Staubli VAL3: home.pjx

--- home.pjx ---
Parameters version=s7.2.1 stackSize=5000 millimeterUnit=true
Program file=changeSession.pgx
Program file=copy_folder.pgx
Program file=isSessionFound.pgx
Program file=loadPage.pgx
Program file=main.pgx
Program file=onEnterEvent.pgx
Program file=onExit.pgx
Program file=onF1Event.pgx
Program file=onF2Event.pgx
Program file=onF3Event.pgx
Program file=onF4Event.pgx
Program file=onF5Event.pgx
Program file=onF6Event.pgx
Program file=onF7Event.pgx
Program file=onF8Event.pgx
Program file=onStart.pgx
Program file=passwd.pgx
Program file=refresh.pgx
Program file=refreshDynamic.pgx
Program file=refreshStatic.pgx
Data file=home.dtx
Library alias=use path=Disk://kernel/userPage/userPage.pjx
Library alias=saveData path=Disk://saveData/saveData.pjx
Library alias=page path=Disk://kernel/template/page/page.pjx
Library alias=language path=Disk://kernel/language/language.pjx
Library alias=processList path=Disk://kernel/processList/processList.pjx
Library alias=cycleStatus path=Disk://cycleStatus/cycleStatus.pjx

--- home.dtx ---
num nKey = 271
public num nPage = 10
num nRefresh = 33.117
num nTime = 1
num nValue[4]
  [0] = 1
  [1] = 2
  [2] = 3
  [3] = 4
public string sItems
string sMenu
string sMessage
string sVersion = "valClean 7.3.1.8"
string sMenu8[8]
string sSession
string sPathSession
string sDeeperSession
bool bButton[8]
  [0] = true
  [1] = true
  [2] = true
  [4] = true
  [5] = true
  [6] = true
  [7] = true

--- main.pgx ---
public program main()
  local bool l_bExit
begin
  // INIT
  call onStart()
  // LOOP UNTIL Exit
  l_bExit=false
  do
    // call the refresh
    call refresh()
    // take the key
    nKey=getKey()
    switch nKey
      case 271
        // select program
        call onF1Event()
      break
      case 272
        // input output
        call onF2Event()
      break
      case 273
        // preset
        call onF3Event()
      break
      case 274
        call onF4Event()
      break
      case 275
        // production page
        call onF5Event()
      break
      case 276
        // maintenance
        call onF6Event()
      break
      case 277
        // advance
        call onF7Event()
      break
      case 278
        // exit
        call onF8Event(l_bExit)
      break
      case 270
        call onEnterEvent()
      break
    endSwitch
    //release the resource
    delay(0)
    // check for the resetMOtion
    if !cycleStatus:bCycle and !cycleStatus:bSimulation and !isEmpty()
      //resetMotion()
    endIf
  until l_bExit
  // on Exit
  call onExit()
end

--- changeSession.pgx ---
program changeSession()
  local num l_nIndex
  local num l_nSize
  local bool l_bDone
  local num i
  local num l_nResult
  local string l_sMessage
  local string l_sPaste
  local string l_sEvent
  local string l_sEmpty
  local string l_sSession
  local string l_sButton[2]
  local bool l_bOk
begin
  // init
  //
  // CREATE THE LIST
  //
  // define your list size for default
  // init
  use:nView=0
  do
    //
    cls()
    call use:setSizeList(19,0,19,11)
    call use:setView(false)
    //
    call use:listcreate("Session")
    // show the message
    call language:page(l_sMessage,1030)
    call use:stringToArray(l_sMessage,sMenu)
    sMenu=""
    if saveData:mode==1
      sMenu[6]=""
    endIf
    if saveData:mode>=1
      call use:setMenu(sMenu,true,3)
    endIf
    // clean the string
    l_sEmpty=""
    call use:stringCopy(l_sEmpty,sSession)
    // get the list of session
    call saveData:getListSession(sSession)
    // build the list
    call use:listadd(sSession)
    // update
    call use:listupdate(0)
    // read the list
    l_bDone=false
    do
      // get the item
      nKey=get()
      call use:listevent(nKey,l_nIndex,l_sEvent)
    until nKey==270 or nKey==255 or ((nKey<=278 and nKey>=275)and sMenu[nKey-271]!="")
    //
    switch nKey
      case 275
        // rename
        l_sPaste=l_sEvent
        call isSessionFound(l_sPaste,l_nResult)
        if l_sPaste!="" and l_sPaste!=l_sEvent
          $rename("session/"+l_sEvent,"session/"+l_sPaste)
        endIf
      break
      case 276
        // duplicate
        l_sPaste=l_sEvent
        call isSessionFound(l_sPaste,l_nResult)
        if l_nResult!=-1
          // duplicate all the file
          call copy_folder(l_sEvent,l_sPaste)
          l_bDone=true
        endIf
      break
      case 277
        // delete
        call saveData:getSession(l_sSession)
        if l_sEvent!=l_sSession and l_sEvent!="default"
          // delete
          call language:getYesNo(l_sButton)
          call language:message(l_sMessage,80)
          l_sMessage=l_sMessage+l_sEvent
          call use:yes_no(l_sMessage,l_sButton,l_bOk)
          if l_bOk
            $delete("Disk://session/"+l_sEvent)
          endIf
        else
          call language:message(l_sMessage,23)
          l_sMessage=l_sMessage+l_sEvent
          popUpMsg(l_sMessage)
        endIf
      break
      case 278
        // create a new one
        // look inside
        call isSessionFound(l_sPaste,l_nResult)
        if l_nResult!=-1
          // create a new one
          call copy_folder("",l_sPaste)
        endIf
      break
    endSwitch
  until l_bDone or nKey==255 or nKey==270
  //
  if nKey!=255 and cycleStatus:bCycle==false and cycleStatus:bSimulation==false
    // check if l_sPaste has been used
    if l_sPaste!=""
      l_sEvent=l_sPaste
    endIf
    // change session
    call language:message(l_sMessage,19)
    l_sMessage=l_sMessage+" SESSION DATA..."
    call use:timerDialog(l_sMessage,0)
      // load the new session
    call saveData:changeSession(l_sEvent)
    // reload the processList using the default saveCycle
    call processList:loadProcessList(i)
    // reset the homing trajectory
    cycleStatus:bHomeLoaded=false
    // save the session
    saveData:libSave()
  endIf
  //
  call use:nullKey(nKey)
end

--- copy_folder.pgx ---
program copy_folder(string x_sPathCopy, string x_sPathPaste)
  local string l_sPathCopy
  local string l_sPathPaste
  local bool l_bCheck
  local num i
  local num j
  local string l_sEmpty
begin
  //
  // copy or not the x_sPathCopy to x_sPath
  //
  call use:timerDialog("Copying file: ##",0)
  call use:stringCopy(l_sEmpty,sPathSession)
  // all the folder are created
  if x_sPathCopy==""
    // copy from the template session
    l_sPathCopy="Disk://kernel/template/session/"
  else
    // copy form the x_sPathCopy session name
    l_sPathCopy="Disk://session/"+x_sPathCopy+"/"
  endIf
  // scan it
  l_bCheck=libList(l_sPathCopy,sPathSession)
  // copy form the x_sPathCopy session name
  l_sPathPaste="Disk://session/"+x_sPathPaste+"/"
  // start the copy
  for i=0 to size(sPathSession)-1
    // for all the directory found only one level...
    l_sEmpty=""
    call use:stringCopy(l_sEmpty,sDeeperSession)
    // scan the folder
    l_bCheck=libList(l_sPathCopy+sPathSession[i],sDeeperSession)
    for j=0 to size(sDeeperSession)-1
      // copy all the file
      call use:typeLen(1,6,l_sPathCopy+sPathSession[i]+"/"+sDeeperSession[j],38)
      call use:typeLen(1,7,l_sPathPaste+sPathSession[i]+"/"+sDeeperSession[j],38)
      l_bCheck=$copy(l_sPathCopy+sPathSession[i]+"/"+sDeeperSession[j],l_sPathPaste+sPathSession[i]+"/"+sDeeperSession[j])
      delay(0)
    endFor
    delay(0)
  endFor
end

--- isSessionFound.pgx ---
program isSessionFound(string& x_sName[], num& x_nResult[])
  local string l_sString
  local bool l_bFound
  local num l_nX
  local num l_nY
  local num i
  local string l_sMessage
begin
  // look if the trajectory already exist
  call language:message(l_sString,21)
  call use:timerDialog(l_sString,0)
  l_nX=(40-len(l_sString))/2
  l_nY=5
  // read the sessino list
  call use:read(l_nX+len(l_sString),l_nY,x_sName,10,false)
  // look for the special char . and /
  if find(x_sName,".")==-1 and find(x_sName,"/")==-1 and find(x_sName,"*")==-1 and find(x_sName,"?")==-1 and find(x_sName,":")==-1 and find(x_sName,chr(34))==-1 and find(x_sName,"\")==-1
    if !use:bUseEscape
      // search inside the sSession
      for i=0 to size(sSession)-1
        if x_sName==sSession[i]
          // trajectory already exist
          call language:message(l_sString,-2)
          popUpMsg(l_sString)
          x_nResult=-1
          return
        endIf
      endFor
    else
      x_nResult=-1
    endIf
  else
    x_nResult=-1
    call language:message(l_sMessage,-3)
    l_sMessage=l_sMessage+" . / * ? : \ "+ chr(34)+" "
    popUpMsg(l_sMessage)
  endIf
end

--- loadPage.pgx ---
program loadPage(string x_sPage, string& x_sItems[])
// load the next page
  local num i
  local string l_sMessage
  local num l_nClock
begin
  // look if the page libload is correct
  i=page:libLoad(x_sPage)
  delay(0)
  if i!=0
    logMsg("[KERNEL] INTERFACE:PAGE LIBLOAD "+x_sPage+" result "+toString("",i))
    call language:message(l_sMessage,-7)
    popUpMsg(l_sMessage+x_sPage+" ; "+toString("",i))
  else
    // copy all the field from x_sItems to the next page
    call use:stringCopy(x_sItems,page:sItems)
    call page:main()
    // to give back
    call use:stringCopy(page:sItems,x_sItems)
  endIf
end

--- onExit.pgx ---
program onExit()
begin
  //
  //  Kill it
  //
  // relaod the template session
  call saveData:changeSession("template")
  // exit
  logMsg("[KERNEL] INTERFACE:Quit")
  cycleStatus:nInterfaceToSV=1
  //
  //
end

--- onF1Event.pgx ---
program onF1Event()
  local num i
  local string l_sItem
  local string l_sPage
begin
  // look if the bButton is enable
  if bButton[0]
    //
    // load Select Program
    l_sPage="Disk://instruction/PROG/page_program"
    l_sItem=""
    call loadPage(l_sPage,l_sItem)
    //
    logMsg("[KERNEL] INTERFACE:PAGE Home Page")
  endIf
end

--- onF2Event.pgx ---
program onF2Event()
  local string l_sItem
  local string l_sPage
begin
  // look if the bButton is enable
  if bButton[1]
    //
    //
    l_sPage="trajectory/page_trajectory"
    call loadPage(l_sPage,l_sItem)
    logMsg("[KERNEL] INTERFACE:PAGE Home Page")
  endIf
end

--- onF3Event.pgx ---
program onF3Event()
  local string l_sItem
  local string l_sPage
begin
  // look if the bButton is enable
  if bButton[2]
    //
    l_sPage="Disk://instruction/inputOutput/page_inOut"
    call loadPage(l_sPage,l_sItem)
    //
    logMsg("[KERNEL] INTERFACE:PAGE Home Page")
  endIf
end

--- onF4Event.pgx ---
program onF4Event()
  local num i
  local string l_sMessage
  local string l_sPage
  local string l_sItem
begin
  // look if the bButton is enable
  if bButton[3]
    l_sPage="Disk://goHome/page_home_set"
    call loadPage(l_sPage,l_sItem)
    logMsg("Disk://goHome/page_home_set")
  endIf
end

--- onF5Event.pgx ---
program onF5Event()
  local string l_sPage
  local string l_sItem
begin
  // look if the bButton is enable
  if bButton[4]
    // LOAD THE CYCLE PAGE
    l_sPage="kernel/page/production"
    call loadPage(l_sPage,l_sItem)
    //
    logMsg("[KERNEL] INTERFACE:PAGE Home Page")
    //
  endIf
end

--- onF6Event.pgx ---
program onF6Event()
  local string l_sItem
  local string l_sPage
begin
  // look if the bButton is enable
  if bButton[5]
    //
    //
    l_sPage="kernel/page/frame"
    call loadPage(l_sPage,l_sItem)
    logMsg("[KERNEL] INTERFACE:PAGE Home Page")
  endIf
end

--- onF7Event.pgx ---
program onF7Event()
  local num local1
  local string l_sPage
  local string l_sItem
begin
  // look if the bButton is enable
  if bButton[6]
    //
    if saveData:mode==0
      call passwd()
      call use:nullKey(nKey)
    else
      l_sPage="Disk://kernel/page/advance"
      call loadPage(l_sPage,l_sItem)
      logMsg("[KERNEL] INTERFACE:PAGE Home Page")
    endIf
  endIf
end

--- onF8Event.pgx ---
program onF8Event(bool& x_bExit[])
  local string l_sMessage
  local string l_sButton[2]
  local num l_nIndex
  local string l_sEvent
  local num l_nKey
  local string l_sItem
begin
  // look if the bButton is enable
  if bButton[7]
    //
    // EXIT or change Session
    //
    if saveData:bMultiSession and saveData:mode>=1
      // init
      use:nView=0
      // ask to change session or quit valplast
      call use:clear(0,13)
      call use:typeMenu(8,"<-")
      call use:setSizeList(30,9,8,2)
      call use:listcreate("")
      l_sItem="Quit"
      call use:listadd(l_sItem)
      l_sItem="Session"
      call use:listadd(l_sItem)
      call use:listupdate(0)
      // loop for a response
      do
        // read a key
        l_nKey=get()
        call use:listevent(l_nKey,l_nIndex,l_sEvent)
      until l_nKey==255 or l_nKey==270
      //
      if l_nKey!=255
        switch l_nIndex
          case 0
            //quit
            // clear the screen
            cls()
            // ask if the user want change the sesion
            call language:message(l_sMessage,4)
            // get the yes_no button Key
            call language:getYesNo(l_sButton)
            // ask the question
            call use:yes_no(l_sMessage,l_sButton,x_bExit)
          break
          case 1
            // change session
            call changeSession()
          break
        endSwitch
      endIf
    elseIf saveData:bMultiSession and saveData:mode==0
      call changeSession()
    else
      // ask if the user want change the sesion
      call language:message(l_sMessage,4)
      // get the yes_no button Key
      call language:getYesNo(l_sButton)
      // ask the question
      call use:yes_no(l_sMessage,l_sButton,x_bExit)
    endIf
  endIf
end

--- onStart.pgx ---
program onStart()
  local num i
  local string l_sMessage
begin
  // wait the START
  wait(cycleStatus:nInterfaceToSV==-1)
  cls()
  //
  setTextMode(0)
  // INIT
  if saveData:mode<2
    userPage(true)
  else
    userPage(false)
  endIf
  //
  logMsg("[KERNEL] INTERFACE:PAGE Home Page, version: " +sVersion)
  //
  // init the session
  // change session
  call language:message(l_sMessage,19)
  l_sMessage=l_sMessage+" SESSION DATA..."
  call use:timerDialog(l_sMessage,0)
  call saveData:changeSession(saveData:sSession)
  call processList:loadProcessList(i)
  // continue
  use:bUseRefresh=true
end

--- passwd.pgx ---
program passwd()
  local string l_sText
  local string l_sTemp
  local num i
  local string l_sMessage
begin
  cls()
  call language:message(l_sMessage,204)
  call use:timerDialog(l_sMessage,0)
  call use:type(2,8,">")
  call use:read(3,8,l_sText,15,true)
  //
  // there are 3 difference kind of access
  // mode 0   ->operator
  // mode 1   ->programmer
  // mode 2   ->integrator
  // mode 3   ->toneage (Administrator)
  //
  saveData:mode=0
  for i=0 to (size(saveData:passwd)-1)
    if l_sText==saveData:passwd[i]
      saveData:mode=i+1
      call use:type(20,8,"...OK...")
      delay(1)
      logMsg("[KERNEL] INTERFACE:Set password to: "+l_sText)
    endIf
  endFor
  if saveData:mode==0
    logMsg("[KERNEL] INTERFACE:Set password to: Operator")
  endIf
  //
  // It's possible to change the password
  //
  if saveData:mode>0 and saveData:mode<3
    call language:message(l_sMessage,205)
    call use:type(0,10,l_sMessage)
    call language:message(l_sMessage,206)
    call use:typeMenu(5,l_sMessage)
    call use:typeMenu(8,"OK")
    nKey=get()
    if nKey==275
      cls()
      call language:message(l_sMessage,207)
      call use:timerDialog(l_sMessage,0)
      call use:type(2,8,">")
      l_sText=""
      call use:read(3,8,l_sText,15,true)
      call language:message(l_sMessage,208)
      call use:timerDialog(l_sMessage,0)
      l_sTemp=""
      call use:read(3,8,l_sTemp,15,true)
      if l_sText==l_sTemp and l_sText!=""
        saveData:passwd[saveData:mode-1]=l_sText
      else
        call language:message(l_sMessage,209)
        popUpMsg(l_sMessage)
      endIf
    endIf
  endIf
  //
  //  Show your mode to access and set the Userpage
  //
  switch saveData:mode
    case 0
      call language:message(l_sText,210)
    break
    case 1
      call language:message(l_sText,211)
    break
    case 2,3
      call language:message(l_sText,212)
    break
  endSwitch
  if saveData:mode<2
    userPage(true)
  else
    userPage(false)
  endIf
  call language:message(l_sMessage,213)
  popUpMsg(l_sMessage+l_sText)
  // SAVE THE SETTING
  saveData:libSave()
end

--- refreshStatic.pgx ---
program refreshStatic()
  local string l_sMessage[2]
  local string l_sMenu
  local string l_sSession
begin
  cls()
  //
  // set the view of the HOME page
  //
  use:nPage=10
  // USE <>PROFILE for <>PAGE
  use:nPage=use:nPage+abs(limit(saveData:mode,0,2)-2)
  // is on Cycle
  if cycleStatus:bCycle
    use:nPage=use:nPage+3
  endIf
  //
  l_sMessage=sVersion
  if saveData:language!="japanese"
    // SET THE VIEW OF THE PAGE
    call language:page(l_sMessage,use:nPage)
    // define the menu
    call use:stringToArray(l_sMessage,sMenu)
  else
    // japanese use the array for the menu
    call language:page(sMenu8,use:nPage)
    call use:stringCopy(sMenu8,sMenu)
  endIf
  // set the menu
  call use:setMenu(sMenu,false,3)
  call use:getMenu(sMenu,bButton)
  // set the F8 message as <-
  if saveData:mode==0 and !saveData:bMultiSession
    call use:typeMenu(8," ")
    bButton[7]=false
  elseIf cycleStatus:bCycle==false and cycleStatus:bSimulation==false
    call use:typeMenu(8," <-")
  elseIf cycleStatus:bCycle==true or cycleStatus:bSimulation==true
    call use:typeMenu(8," ")
  endIf
  //
  // show the profile
  //
  call language:message(l_sMessage,5)
  call language:message(l_sMessage[1],limit(saveData:mode,0,2))
  l_sMessage=l_sMessage+":"+l_sMessage[1]
  call use:type(0,0,l_sMessage)
  //
  // show the session name
  //
  call saveData:getSession(l_sSession)
  if l_sSession!=""
    // start on the right
    l_sSession="Session: "+l_sSession
    call use:type(40-len(l_sSession),1,l_sSession)
  endIf
  //
end
